FUNCTION_BLOCK FB_Drive
VAR_INPUT
	b_Enable				: BOOL;		
	b_Reset					: BOOL;
	f_Override				: LREAL;
	b_JogForward			: BOOL;
	b_JogBackwards			: BOOL;
	b_MoveAbsolute			: BOOL;
	n_MoveAbsoluteDirection	: MC_Direction;
	b_Home					: BOOL;
	f_Velocity				: LREAL;
	f_Acceleration			: LREAL;
	f_Deceleration			: LREAL;
	f_Jerk					: LREAL;
	f_Position				: LREAL;
	
END_VAR
VAR_OUTPUT
	b_PowerActive			: BOOL;
	b_Error					: BOOL;
	n_ErrorID				: UDINT;
	b_MoveAbsoluteDone		: BOOL;
	f_ActVelocity			: LREAL;
	f_ActTorque				: LREAL;
	f_ActPosition			: LREAL;
END_VAR
VAR_IN_OUT
	Axis					: AXIS_REF;
END_VAR
VAR
	fb_MC_Reset				: MC_Reset;
	fb_MC_Power				: MC_Power;
	fb_MC_SetPosition		: FB_SoEAX5000SetPositionOffset;
	fb_MC_Halt				: MC_Halt;
	fb_MC_Jog				: MC_Jog;
	fb_MC_Absolute			: MC_MoveModulo;
END_VAR

//***********************************************************************************
//
// ETH Zürich / Robotic Fabrication Lab
// HIB C 13 / Stefano-Franscini-Platz 1
// CH-8093 Zürich
// 
// ***********************************************************************************
// 
// PROJECT     :  ?? 
// 
// FUNCTION    :  General Function Block for Drives 
// 
// AUTHOR      :  Mathias Suter
// 
// EMAIL       :  mathias.suter@solinaut.ch
// 
// Copyright   :  ETH Zürich (CH) 2021
//
// ***********************************************************************************


//
// Axis Power
fb_MC_Power(
	Axis			:= Axis,    
	Enable          := b_Enable,
    Enable_Positive := b_Enable, 
    Enable_Negative := b_Enable,
    Override        := f_Override);
	
//
// Axis Stop
fb_MC_Halt(
	Axis			:= Axis,
	Execute			:= NOT b_enable,
	Deceleration	:= 1000);
	

//
// Axis Reset	
fb_MC_Reset(
	Axis			:= Axis,    
	Execute         := b_Reset);
	
//
// Axis SetPosition
(*fb_MC_SetPosition(
	Axis			:= Axis,    
	Execute         := b_Home,
	Position		:= f_Position);*)
	
	
fb_MC_SetPosition(
	Axis			:= Axis,    
	Execute         := b_Home,
	memory			:= 1,
	Feedback		:= 0,
	Position		:= f_Position);
	
//
// Axis Jog
fb_MC_Jog(
	Axis			:= Axis,    
	JogForward      := b_JogForward AND fb_MC_Power.Status AND b_Enable,
    JogBackwards 	:= b_JogBackwards AND fb_MC_Power.Status AND b_Enable, 
    Mode 			:= MC_JOGMODE_CONTINOUS,
    Velocity        := f_Velocity,
	Acceleration	:= f_Acceleration,
	Deceleration	:= f_Deceleration,
	Jerk			:= f_Jerk);

//
// Axis Absolute	
fb_MC_Absolute(
	Axis			:= Axis,
	Execute			:= b_MoveAbsolute AND b_Enable,
	Position		:= f_Position,
	Velocity		:= f_Velocity,
	Acceleration	:= f_Acceleration,
	Jerk			:= f_Jerk,
    Direction		:= n_MoveAbsoluteDirection);
	
	
//
// Ouptut Power Active
b_PowerActive := fb_MC_Power.Status;	
	
// Output MoveAbsoluteDone
b_MoveAbsoluteDone := fb_MC_Absolute.Done;

//
// Output Actual Velocity, Torque, Position
f_ActVelocity := Axis.NcToPlc.ActVelo;
f_ActTorque	:= Axis.NcToPlc.ActTorque;
f_ActPosition := Axis.NcToPlc.ModuloActPos;	
		
//
// Output Error
b_Error := fb_MC_Power.Error OR fb_MC_Reset.Error OR fb_MC_SetPosition.Error OR fb_MC_Jog.Error OR fb_MC_Absolute.Error;

//
// Output ErrorID
IF fb_MC_Power.Error THEN
	n_ErrorID := fb_MC_Power.ErrorID;
ELSIF fb_MC_Reset.Error THEN
	n_ErrorID := fb_MC_Reset.ErrorID;
ELSIF fb_MC_SetPosition.Error THEN
	n_ErrorID := fb_MC_SetPosition.ErrorID;
ELSIF fb_MC_Jog.Error THEN
	n_ErrorID := fb_MC_Jog.ErrorID;
ELSIF fb_MC_Absolute.Error THEN
	n_ErrorID := fb_MC_Absolute.ErrorID;
ELSE
	n_ErrorID := 0;	
END_IF;

END_FUNCTION_BLOCK

(* stored: Version 1.1.0.1, ProductVersion 3.1.4024.4
   POU FB_Drive: Id {b7fbeb4c-85cf-401d-b15a-e5632b281c02}, SpecialFunc None *)
